  [1275] = {j1=-11.226, j2=60.578, j3=50.227, j4=-2.907, j5=77.416, j6=-7.201}
  [1276] = {j1=-11.247, j2=60.183, j3=50.546, j4=-2.858, j5=77.210, j6=-7.506}
  [1277] = {j1=-11.262, j2=59.787, j3=50.867, j4=-2.835, j5=77.009, j6=-7.789}
  [1278] = {j1=-11.270, j2=59.393, j3=51.185, j4=-2.836, j5=76.815, j6=-8.050}
  [1279] = {j1=-11.270, j2=59.003, j3=51.497, j4=-2.860, j5=76.631, j6=-8.287}
  [1280] = {j1=-11.271, j2=58.982, j3=51.520, j4=-2.860, j5=76.610, j6=-8.296}
  [1281] = {j1=-11.272, j2=59.014, j3=51.464, j4=-2.853, j5=76.694, j6=-8.234}
  [1282] = {j1=-11.273, j2=59.020, j3=51.466, j4=-2.850, j5=76.684, j6=-8.227}
  [1283] = {j1=-11.273, j2=59.395, j3=51.183, j4=-2.823, j5=76.835, j6=-7.992}
  [1284] = {j1=-11.267, j2=59.773, j3=50.893, j4=-2.818, j5=76.995, j6=-7.734}
  [1285] = {j1=-11.253, j2=60.153, j3=50.600, j4=-2.838, j5=77.163, j6=-7.453}
  [1286] = {j1=-11.233, j2=60.534, j3=50.307, j4=-2.884, j5=77.337, j6=-7.150}
  [1287] = {j1=-11.206, j2=60.969, j3=49.972, j4=-2.950, j5=77.543, j6=-6.787}
  [1288] = {j1=-11.181, j2=61.404, j3=49.637, j4=-3.012, j5=77.758, j6=-6.420}
  [1289] = {j1=-11.158, j2=61.840, j3=49.301, j4=-3.068, j5=77.985, j6=-6.048}
  [1290] = {j1=-11.138, j2=62.278, j3=48.960, j4=-3.118, j5=78.224, j6=-5.671}
  [1291] = {j1=-11.121, j2=62.719, j3=48.611, j4=-3.159, j5=78.479, j6=-5.288}
  [1292] = {j1=-11.107, j2=63.165, j3=48.253, j4=-3.190, j5=78.752, j6=-4.899}
  [1293] = {j1=-11.096, j2=63.618, j3=47.883, j4=-3.210, j5=79.045, j6=-4.504}
  [1294] = {j1=-11.095, j2=63.691, j3=47.828, j4=-3.212, j5=79.084, j6=-4.434}
  [1295] = {j1=-11.072, j2=64.145, j3=47.454, j4=-3.279, j5=79.386, j6=-4.006}
  [1296] = {j1=-11.021, j2=64.658, j3=47.052, j4=-3.457, j5=79.694, j6=-3.472}
  [1297] = {j1=-10.947, j2=65.119, j3=46.749, j4=-3.736, j5=79.878, j6=-2.955}
  [1298] = {j1=-10.881, j2=65.440, j3=46.609, j4=-3.998, j5=79.892, j6=-2.594}
  [1299] = {j1=-10.822, j2=65.711, j3=46.557, j4=-4.248, j5=79.794, j6=-2.311}
  [1300] = {j1=-10.766, j2=65.940, j3=46.579, j4=-4.492, j5=79.599, j6=-2.093}
  [1301] = {j1=-10.713, j2=66.134, j3=46.661, j4=-4.735, j5=79.323, j6=-1.928}
  [1302] = {j1=-10.661, j2=66.298, j3=46.792, j4=-4.981, j5=78.981, j6=-1.805}
  [1303] = {j1=-10.609, j2=66.438, j3=46.958, j4=-5.235, j5=78.590, j6=-1.712}
  [1304] = {j1=-10.609, j2=66.450, j3=46.937, j4=-5.235, j5=78.635, j6=-1.666}
  [1305] = {j1=-10.662, j2=66.295, j3=46.797, j4=-4.977, j5=78.990, j6=-1.761}
  [1306] = {j1=-10.715, j2=66.116, j3=46.694, j4=-4.727, j5=79.294, j6=-1.885}
  [1307] = {j1=-10.769, j2=65.906, j3=46.639, j4=-4.480, j5=79.533, j6=-2.052}
  [1308] = {j1=-10.826, j2=65.661, j3=46.646, j4=-4.231, j5=79.692, j6=-2.272}
  [1309] = {j1=-10.887, j2=65.374, j3=46.726, j4=-3.975, j5=79.754, j6=-2.556}
  [1310] = {j1=-10.954, j2=65.038, j3=46.895, j4=-3.709, j5=79.705, j6=-2.918}
  [1311] = {j1=-11.030, j2=64.561, j3=47.225, j4=-3.424, j5=79.488, j6=-3.436}
  [1312] = {j1=-11.082, j2=64.032, j3=47.654, j4=-3.241, j5=79.147, j6=-3.969}
  [1313] = {j1=-11.106, j2=63.563, j3=48.056, j4=-3.171, j5=78.810, j6=-4.398}
  [1314] = {j1=-11.109, j2=63.474, j3=48.140, j4=-3.165, j5=78.734, j6=-4.468}
  [1315] = {j1=-11.121, j2=63.004, j3=48.541, j4=-3.141, j5=78.405, j6=-4.864}
  [1316] = {j1=-11.137, j2=62.540, j3=48.931, j4=-3.105, j5=78.094, j6=-5.254}
  [1317] = {j1=-11.156, j2=62.080, j3=49.312, j4=-3.060, j5=77.799, j6=-5.639}
  [1318] = {j1=-11.177, j2=61.623, j3=49.688, j4=-3.006, j5=77.520, j6=-6.019}
  [1319] = {j1=-11.201, j2=61.168, j3=50.059, j4=-2.945, j5=77.254, j6=-6.394}
  [1320] = {j1=-11.228, j2=60.714, j3=50.428, j4=-2.879, j5=76.998, j6=-6.764}
  [1321] = {j1=-11.257, j2=60.260, j3=50.797, j4=-2.808, j5=76.752, j6=-7.128}
  [1322] = {j1=-11.279, j2=59.860, j3=51.124, j4=-2.757, j5=76.541, j6=-7.433}
  [1323] = {j1=-11.294, j2=59.462, j3=51.450, j4=-2.733, j5=76.335, j6=-7.715}
  [1324] = {j1=-11.303, j2=59.065, j3=51.774, j4=-2.733, j5=76.137, j6=-7.973}
  [1325] = {j1=-11.304, j2=58.671, j3=52.092, j4=-2.756, j5=75.948, j6=-8.207}
  [1326] = {j1=-11.305, j2=58.646, j3=52.122, j4=-2.755, j5=75.918, j6=-8.216}
  [1327] = {j1=-11.117, j2=63.463, j3=48.236, j4=-3.132, j5=78.603, j6=-4.344}
  [1328] = {j1=-11.094, j2=63.912, j3=47.868, j4=-3.198, j5=78.894, j6=-3.918}
  [1329] = {j1=-11.043, j2=64.421, j3=47.475, j4=-3.376, j5=79.188, j6=-3.387}
  [1330] = {j1=-10.968, j2=64.879, j3=47.178, j4=-3.659, j5=79.360, j6=-2.869}
  [1331] = {j1=-10.902, j2=65.198, j3=47.040, j4=-3.923, j5=79.367, j6=-2.505}
  [1332] = {j1=-10.841, j2=65.470, j3=46.987, j4=-4.176, j5=79.263, j6=-2.218}
  [1333] = {j1=-10.785, j2=65.700, j3=47.007, j4=-4.423, j5=79.065, j6=-1.995}
  [1334] = {j1=-10.731, j2=65.896, j3=47.086, j4=-4.668, j5=78.788, j6=-1.824}
  [1335] = {j1=-10.678, j2=66.064, j3=47.211, j4=-4.915, j5=78.446, j6=-1.694}
  [1336] = {j1=-10.626, j2=66.207, j3=47.372, j4=-5.171, j5=78.055, j6=-1.594}
  [1337] = {j1=-10.626, j2=66.222, j3=47.346, j4=-5.172, j5=78.113, j6=-1.532}
  [1338] = {j1=-10.680, j2=66.056, j3=47.225, j4=-4.910, j5=78.450, j6=-1.633}
  [1339] = {j1=-10.734, j2=65.866, j3=47.140, j4=-4.655, j5=78.736, j6=-1.765}
  [1340] = {j1=-10.790, j2=65.647, j3=47.103, j4=-4.404, j5=78.958, j6=-1.938}
  [1341] = {j1=-10.848, j2=65.392, j3=47.127, j4=-4.150, j5=79.100, j6=-2.163}
  [1342] = {j1=-10.911, j2=65.096, j3=47.222, j4=-3.890, j5=79.149, j6=-2.453}
  [1343] = {j1=-10.980, j2=64.753, j3=47.404, j4=-3.617, j5=79.088, j6=-2.818}
  [1344] = {j1=-11.057, j2=64.271, j3=47.743, j4=-3.326, j5=78.863, j6=-3.338}
  [1345] = {j1=-11.111, j2=63.738, j3=48.180, j4=-3.140, j5=78.516, j6=-3.869}
  [1346] = {j1=-11.135, j2=63.264, j3=48.592, j4=-3.068, j5=78.170, j6=-4.296}
  [1347] = {j1=-11.137, j2=63.282, j3=48.560, j4=-3.059, j5=78.230, j6=-4.235}
  [1348] = {j1=-11.115, j2=63.725, j3=48.204, j4=-3.123, j5=78.505, j6=-3.812}
  [1349] = {j1=-11.063, j2=64.226, j3=47.824, j4=-3.303, j5=78.780, j6=-3.284}
  [1350] = {j1=-10.987, j2=64.677, j3=47.538, j4=-3.588, j5=78.933, j6=-2.766}
  [1351] = {j1=-10.920, j2=64.992, j3=47.409, j4=-3.855, j5=78.925, j6=-2.400}
  [1352] = {j1=-10.859, j2=65.260, j3=47.362, j4=-4.110, j5=78.809, j6=-2.109}
  [1353] = {j1=-10.802, j2=65.489, j3=47.386, j4=-4.358, j5=78.601, j6=-1.881}
  [1354] = {j1=-10.748, j2=65.683, j3=47.468, j4=-4.604, j5=78.313, j6=-1.704}
  [1355] = {j1=-10.695, j2=65.849, j3=47.596, j4=-4.853, j5=77.962, j6=-1.568}
  [1356] = {j1=-10.642, j2=65.991, j3=47.759, j4=-5.109, j5=77.560, j6=-1.461}
  [1357] = {j1=-10.643, j2=65.992, j3=47.759, j4=-5.107, j5=77.578, j6=-1.413}
  [1358] = {j1=-10.698, j2=65.811, j3=47.664, j4=-4.840, j5=77.885, j6=-1.520}
  [1359] = {j1=-10.754, j2=65.605, j3=47.608, j4=-4.581, j5=78.139, j6=-1.658}
  [1360] = {j1=-10.812, j2=65.368, j3=47.602, j4=-4.323, j5=78.326, j6=-1.837}
  [1361] = {j1=-10.872, j2=65.094, j3=47.658, j4=-4.062, j5=78.432, j6=-2.068}
  [1362] = {j1=-10.937, j2=64.779, j3=47.789, j4=-3.794, j5=78.440, j6=-2.363}
  [1363] = {j1=-11.008, j2=64.414, j3=48.009, j4=-3.513, j5=78.335, j6=-2.733}
  [1364] = {j1=-11.089, j2=63.908, j3=48.391, j4=-3.211, j5=78.061, j6=-3.256}
  [1365] = {j1=-11.146, j2=63.346, j3=48.881, j4=-3.015, j5=77.650, j6=-3.789}
  [1366] = {j1=-11.174, j2=62.830, j3=49.369, j4=-2.931, j5=77.211, j6=-4.217}
public mdesc mNomSpeed = {accel=100, vel=100, decel=100, tmax=99999, rmax=99999, blend=off, leave=50, reach=50}
public mdesc mdJointBlend = {accel=250, vel=30, decel=150, tmax=99999, rmax=99999, blend=off, leave=0, reach=0}
public mdesc mdLineBlend = {accel=80, vel=30, decel=30, tmax=763.92, rmax=9999, blend=joint, leave=0.1, reach=0.1}
public tool tTool = {x=968.000, y=-155.000, z=-238.000, rx=-90.000, ry=0.000, rz=180.000, fatherId=flange[0], ioLink=valve1}
